FUNCTION_BLOCK Actuator 
VAR_INPUT
END_VAR
VAR_OUTPUT
	fbOutput : BoolOut;
END_VAR
VAR
END_VAR

END_FUNCTION_BLOCK

(* stored: Version 1.1.0.1, ProductVersion 3.1.4024.2
   POU Actuator: Id {bd3f25da-700d-4a57-b9b7-112a23ed66c4}, SpecialFunc None *)
